INTERFACE I_AmrModule EXTENDS I_Module, I_Override, I_ContainStatemachine

PROPERTY BypassScanners : BOOL
SET
END_SET
END_PROPERTY

PROPERTY Lift : I_Axis_PTP
GET
END_GET
END_PROPERTY

METHOD ResetSafety
END_METHOD

PROPERTY WheelLeft : I_Axis_PTP
GET
END_GET
END_PROPERTY

PROPERTY WheelLeftStreamVelocity : I_Navitrol_StreamVelocity
GET
END_GET
END_PROPERTY

PROPERTY WheelRight : I_Axis_PTP
GET
END_GET
END_PROPERTY

PROPERTY WheelRightStreamVelocity : I_Navitrol_StreamVelocity
GET
END_GET
END_PROPERTY

END_INTERFACE

(* stored: Version 1.1.0.1
   Itf I_AmrModule: Id {9169f098-efd6-41e1-afc0-6d9ff7eb0ed9}
   Property BypassScanners: Id {d566d36b-114b-40f2-8f6b-e4a3ca2303e3}
   Set Set: Id {55b94751-aca6-4434-9d1f-0206cf8e4ea4}
   Property Lift: Id {270e6659-b12d-4f79-9298-601355dd78e8}
   Get Get: Id {904335e2-75c1-4137-bfbf-6ce633d9cd9e}
   Method ResetSafety: Id {e0e00371-221d-45c1-b6b2-bf77f57b2c83}
   Property WheelLeft: Id {66ae7755-ec64-4bb3-895f-f309104d0c75}
   Get Get: Id {1807b374-3a18-4b5e-a8b3-004fcf038e51}
   Property WheelLeftStreamVelocity: Id {eafbd0ef-345f-4c82-8272-d8ac2e243871}
   Get Get: Id {8cfb8182-d1a0-414d-8461-a562cd9811a8}
   Property WheelRight: Id {d12793d9-ce17-41bc-a334-ee8282413127}
   Get Get: Id {2980ebb1-8327-4166-a784-7f5c327088fc}
   Property WheelRightStreamVelocity: Id {3c89224c-f66e-45e7-9d3a-49fb63920154}
   Get Get: Id {a377acdd-ff76-4e82-b6b2-ef81c1ceb807} *)
